{attribute 'OPC.UA.DA' := '1'}
FUNCTION_BLOCK FW212CPolarisationFilter EXTENDS PolarisationFilterBase
VAR_INPUT
END_VAR
VAR_OUTPUT
END_VAR
VAR
	{attribute 'OPC.UA.DA' := '0'}
	_config : FW212CPolarisationFilterConfig;
	{attribute 'OPC.UA.DA' := '0'}
	_coeAccess : CoeAccess;
	{attribute 'OPC.UA.DA' := '0'}
	_initConfigSerialCom : BOOL;
	{attribute 'OPC.UA.DA' := '0'}
	_serialCom  : SerialCom(Prefix :='', Suffix := Const.CARRIAGE_RETURN);
	{attribute 'OPC.UA.DA' := '0'}	
	_refSerialCom : REFERENCE TO SerialCom(Prefix :='', Suffix := Const.CARRIAGE_RETURN) := _serialCom; 
	{attribute 'OPC.UA.DA' := '0'}
	_isReceived : BOOL;
	
	{attribute 'OPC.UA.DA' := '0'}
	_deliverMessages : INT;
	
	CheckConnectionMsg : STRING(255);
	PositionMsg : STRING(255);
	PositionCountMsg : STRING(255);
	IdMsg : STRING(255);
	CustomMsg : STRING(255);
	
	{region 'Commands'}
		
	{attribute 'OPC.UA.DA' := '0'}
	_moveAbsPosition     : BOOL;
	{attribute 'OPC.UA.DA' := '0'}
	_jogBackwardPosition : BOOL;
	{attribute 'OPC.UA.DA' := '0'}
	_jogForwardPosition  : BOOL;
	{attribute 'OPC.UA.DA' := '0'}
	_customCmd : BOOL;	
	
	{endregion}
	
	{attribute 'OPC.UA.DA' := '0'}
	_initDevice : BOOL;	
	
	{attribute 'OPC.UA.DA' := '0'}
	_pos : INT;	 
	{attribute 'OPC.UA.DA' := '0'}
	_cmd : STRING;	
	{attribute 'OPC.UA.DA' := '0'}
	_itemScheduler : INT;		
	{attribute 'OPC.UA.DA' := '0'}
	_pulseGenerator : TON;	
			
	{attribute 'OPC.UA.DA' := '0'}
	message : STRING;
	{attribute 'OPC.UA.DA' := '0'}
	_length : INT;
	
END_VAR


IF NOT InitConfigSerialCom THEN
	ConfigureSerialCom();
ELSE
	IF _refSerialCom.ErrorReceiveId = COMERROR_NOERROR THEN
		_refSerialCom(TxBuffer := HardwareGlobalVariables.TxBufferPolarisation, 
		 	      	  RxBuffer := HardwareGlobalVariables.RxBufferPolarisation);
	END_IF	
				  
	// Init device
	InitDevice(); 				  
				  
	// Deliver messages
	IF _refSerialCom.IsReceived THEN
		CASE _deliverMessages OF			
			EFeedbackMsgPolarisationFW212C.CheckConnectionMsg :
				CheckConnectionMsg := _refSerialCom.LastReceivedString;	
			EFeedbackMsgPolarisationFW212C.PositionMsg :
				PositionMsg := _refSerialCom.LastReceivedString;
			EFeedbackMsgPolarisationFW212C.PositionCountMsg :
				PositionCountMsg := _refSerialCom.LastReceivedString;
			EFeedbackMsgPolarisationFW212C.IdMsg :
				IdMsg := _refSerialCom.LastReceivedString;
			EFeedbackMsgPolarisationFW212C.CustomMsg :
				CustomMsg := _refSerialCom.LastReceivedString;						
		END_CASE
		
		_deliverMessages := 0;
	END_IF							   							   		
END_IF

IF InitConfigSerialCom THEN			
	MoveAbsPosition(_moveAbsPosition, _pos);	
	JogBackwardPosition(_jogBackwardPosition);				
	JogForwardPosition(_jogForwardPosition);
	CustomCommand(_customCmd, _cmd);	

	IF (NOT _moveAbsPosition AND NOT _jogBackwardPosition AND NOT _jogForwardPosition AND NOT _customCmd) THEN
		MessageScheduler();
	END_IF	
END_IF

METHOD CheckConnection
VAR_INPUT
END_VAR
VAR
	cmd : STRING := '';
END_VAR
_deliverMessages := EFeedbackMsgPolarisationFW212C.CheckConnectionMsg;
_serialCom.Send(cmd);
END_METHOD

METHOD ConfigureSerialCom
VAR_INPUT
END_VAR
IF _coeAccess.CoeOperation.Ready THEN
	_logger.Information(_message.Reset().Append('Start configuration com serial').ToString());
END_IF;	

_coeAccess.CoeOperation.Start();
_coeAccess(SerialCommunication := _config.SerialCommunication);
	
IF _coeAccess.CoeOperation.Done THEN
	_coeAccess.SetDone();
	
	_Logger.Information(_message.Reset().
							Append('{').Append(TO_STRING(THIS^.Family)).Append('} : ').
							Append(' - Status : ').Append(TO_STRING(_coeAccess.Status)).ToString());	
	InitConfigSerialCom := TRUE;
END_IF
 
IF _coeAccess.CoeOperation.Error THEN	
	_coeAccess.SetError(0);
	
	_Logger.Error(_message.Reset().
							Append('{').Append(TO_STRING(THIS^.Family)).Append('} : ').
							Append(' - Status : ').Append(TO_STRING(_coeAccess.Status)).ToString());	
	InitConfigSerialCom := TRUE;
END_IF

THIS^.Status := _coeAccess.Status;
State := _coeAccess.Status;
END_METHOD

{attribute 'TcRpcEnable' := '1'}
METHOD CustomCommand
VAR_INPUT
	Execute : BOOL;
	Cmd : STRING;
END_VAR
IF Execute THEN
	_logger.Information(_message.Reset().
								Append(_config.Name).
								Append(' - Custom : ').
								Append(Cmd).ToString());	
	_deliverMessages := EFeedbackMsgPolarisationFW212C.CustomMsg;								
	_serialCom.Send(Cmd);
	
	_customCmd := FALSE;
END_IF
END_METHOD

METHOD FB_init : BOOL
VAR_INPUT
	bInitRetains : BOOL; // if TRUE, the retain variables are initialized (warm start / cold start)
	bInCopyCode : BOOL;  // if TRUE, the instance afterwards gets moved into the copy code (online change)
	Config : FW212CPolarisationFilterConfig;
END_VAR
IF Config.IsEnabled THEN
	_config := Config;
	
	SUPER^._polarisationFilterConfig.Name := Config.Name;
	SUPER^._polarisationFilterConfig.DeviceID := Config.DeviceID;
	SUPER^._polarisationFilterConfig.IsEnabled := Config.IsEnabled;
	SUPER^._polarisationFilterConfig.LogLevel := Config.LogLevel;
	
	SUPER^.Name := Config.Name;
	SUPER^.DeviceID := Config.DeviceID;	
	THIS^.Family := DeviceFamily.PolarisationFilter;
	
	_Logger.Information(_message.Reset().Append('Init ').
							Append('{').Append(TO_STRING(THIS^.Family)).Append('} - ').
							Append('{').Append(TO_STRING(Config.Name)).Append('}').ToString());																													
END_IF
END_METHOD

(** Returns the model number and firmware version **)
METHOD GetIdentifier : STRING
VAR_INPUT
END_VAR
VAR
	cmd : STRING := '*idn?';
END_VAR
_deliverMessages := EFeedbackMsgPolarisationFW212C.IdMsg;
_serialCom.Send(cmd);
END_METHOD

(** Position Query **)
METHOD PROTECTED GetPosition 
VAR_INPUT
END_VAR
VAR
	cmd : STRING := 'pos?';
END_VAR
_deliverMessages := EFeedbackMsgPolarisationFW212C.PositionMsg;
_serialCom.Send(cmd);
END_METHOD

(** Returns the wheel type **)
METHOD GetPositionCount
VAR_INPUT
END_VAR
VAR
	cmd : STRING := 'pcount?';
END_VAR
_deliverMessages := EFeedbackMsgPolarisationFW212C.PositionCountMsg;
_serialCom.Send(cmd);
END_METHOD

PROPERTY InitConfigSerialCom : BOOL
GET
InitConfigSerialCom := _initConfigSerialCom;
END_GET
SET
_initConfigSerialCom := InitConfigSerialCom;
END_SET
END_PROPERTY

METHOD InitDevice
VAR_INPUT
END_VAR
IF NOT _initDevice THEN	
	_logger.Information(_message.Reset().
								Append(_config.Name).
								Append(' - Init device').ToString());

	// TODO : define max count 
	
	_initDevice := TRUE;	
END_IF
END_METHOD

{attribute 'TcRpcEnable' := '1'}
(** Decrements the filter position by 1 **)
METHOD PROTECTED JogBackwardPosition
VAR_INPUT
	Execute : BOOL;
END_VAR
VAR
	DecFilterPos : BYTE := 68;
	posArray     : ARRAY[1..3] OF BYTE := [27, 91, DecFilterPos];
END_VAR
IF Execute THEN
	_logger.Information(_message.Reset().
								Append(_config.Name).
								Append(' - Jog backward position').ToString());
	_serialCom.Send3B(posArray);
	_jogBackwardPosition := FALSE;
END_IF
END_METHOD

{attribute 'TcRpcEnable' := '1'}
(** Increments the filter position by 1 **)
METHOD PROTECTED JogForwardPosition
VAR_INPUT
	Execute : BOOL;
END_VAR
VAR
	jogForwardPos : BYTE := 67;
	posArray     : ARRAY[1..3] OF BYTE := [27, 91, jogForwardPos];
END_VAR
IF Execute THEN
	_logger.Information(_message.Reset().
								Append(_config.Name).
								Append(' - Jog forward position').ToString());
	_serialCom.Send3B(posArray);
	_jogForwardPosition := FALSE;
END_IF
END_METHOD

METHOD MessageScheduler
VAR_INPUT
END_VAR
IF _pulseGenerator.Q THEN
	_pulseGenerator(IN := FALSE, PT := T#10MS);
		
	CASE _itemScheduler OF
		0:  GetIdentifier();
			_itemScheduler := 1;

		1:	GetPosition();
			_itemScheduler := 2;
			
		2:  GetPositionCount();
			_itemScheduler := 3;
			
		3:  CheckConnection();
			_itemScheduler := 0;								
	END_CASE
ELSE
	_pulseGenerator(IN := TRUE, PT := T#50MS);	
END_IF
END_METHOD

{attribute 'TcRpcEnable' := '1'}
(** Moves the wheel to filter position n **)
METHOD PROTECTED MoveAbsPosition
VAR_INPUT
	Execute : BOOL;
	Position : LREAL;
END_VAR
VAR
	cmd : STRING := 'pos=';
END_VAR
IF Execute THEN
	_logger.Information(_message.Reset().
								Append(_config.Name).
								Append(' - Move absolute position : ').Append(TO_STRING(Position)).ToString());
	_serialCom.Send(CONCAT(cmd, TO_STRING(Position)));
	_moveAbsPosition := FALSE;
END_IF
END_METHOD

{attribute 'TcRpcEnable' := '1'}
METHOD RaisePropertiesChanged
VAR_INPUT
	Execute : BOOL;
END_VAR
IF Execute THEN
	CheckConnectionMsg := ' ';
	PositionMsg := ' ';
	IdMsg := ' ';
	CustomMsg := ' ';
END_IF
END_METHOD

END_FUNCTION_BLOCK

(* stored: Version 1.1.0.1, ProductVersion 3.1.4024.12
   POU FW212CPolarisationFilter: Id {ff9e6a1d-f467-403a-ae33-bac95d4ebb11}, SpecialFunc None
   Folder Commands: Id {02498fe1-037b-4e7a-8095-ae600a4eac7f}
   Method CheckConnection: Id {0ecc6f1c-2669-4558-972d-b42c8eac2825}
   Method ConfigureSerialCom: Id {1f9898b2-9ec1-4261-a627-98bda2b19de6}
   Method CustomCommand: Id {d8c45193-ca7d-4083-9635-7b290ad8fb6a}
   Method FB_init: Id {3d12d8a4-2b9d-44ce-b7c8-6eb15ad0cebd}
   Method GetIdentifier: Id {659aa7b3-a36a-4f1a-a805-7ca918e413ab}
   Method GetPosition: Id {cb43dfb6-138d-4e8b-8621-4074e0d8c4f1}
   Method GetPositionCount: Id {e48d1370-530e-425e-bb7d-eaa0fcfcc4a3}
   Property InitConfigSerialCom: Id {14f4e0ee-8e30-49e3-a89e-19614b337338}
   Get Get: Id {4c053e10-8d57-49ac-a5f4-dc1e8ae8297a}
   Set Set: Id {3b3c764f-6536-4ed2-a0b1-b7cec589de65}
   Method InitDevice: Id {084a1bc3-a8d6-4aa3-ad26-23754f27bafc}
   Method JogBackwardPosition: Id {6bfc15cc-9c7d-4f07-a05f-77706cdd9ed5}
   Method JogForwardPosition: Id {72316f18-fceb-4771-a6b8-f7fd8ba702e4}
   Method MessageScheduler: Id {94b75cfd-9e5e-49a8-a1a3-7bbd319f5321}
   Method MoveAbsPosition: Id {56e5996d-f845-41f2-a3db-95b5baf40e4b}
   Method RaisePropertiesChanged: Id {9951505e-bde0-4233-b7ac-c6b72c97ee87} *)
